RoboDK station: Example-03.b-Welding Station - Fanuc.rdk

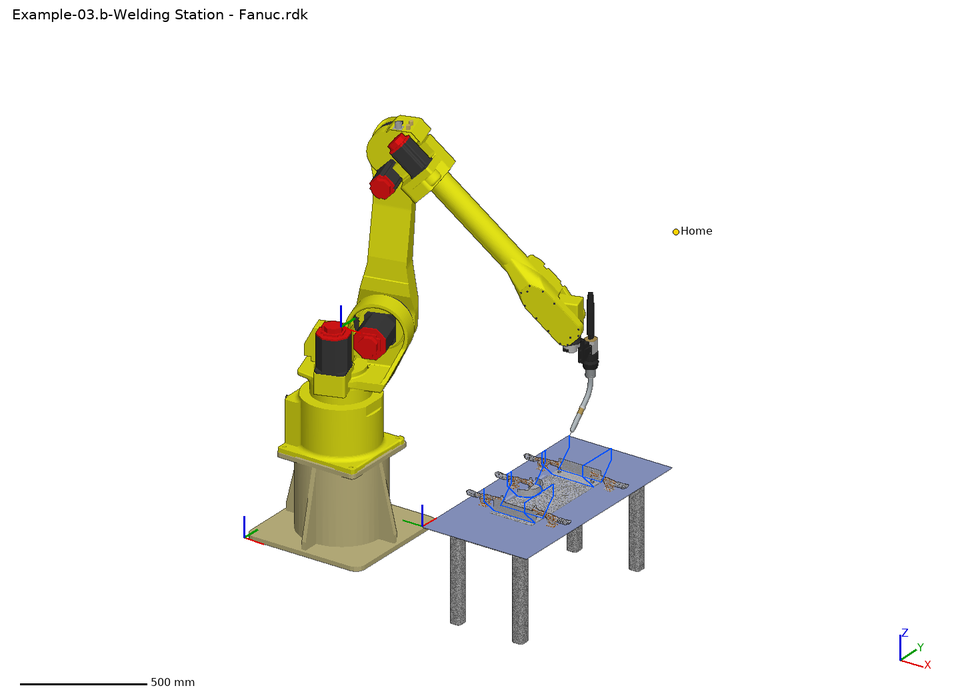
[picture v0: the station drawn from its stored meshes, robots at their saved joint values, targets as dots, program paths as lines]
Station Ex 01 - Fanuc Welding Station (saved by RoboDK 5.2.3). Poses are relative to the parent item; angles as X-Y-Z fixed-axis rotations.
Station parameters (name, value as stored): Torch1, 4, red, 0
  - frame Fanuc ARC Mate 120iB/10L Base at (0, 0, 525) mm
    - robot Fanuc ARC Mate 120iB/10L: 6 axes, payload 10 kg, reach 1885 mm, repeatability 0.1 mm, weight 225 kg
        modified DH rows (alpha deg, a mm, theta deg, d mm): 0, 0, 0, 525; -90, 150, -90, 0; 0, 770, 0, 0; -90, 100, 0, 960; 90, 0, 0, 0; -90, 0, 0, 100
        base shift (0, 0, -525) mm
        joint limits [-170, -80, -170, -200, -140, -150] to [170, 170, 250, 200, 140, 450]; home [0, 0, 0, 0, 0, 0]; saved at [18.463, 3.094, -45.099, 0, -44.901, 431.537]
      - tool Daihen OTC weld gun, TCP at (-2, 0, 402) mm, rotated rx 0 ry 45 rz 180 deg, size 201.6 x 65.1 x 567.7 mm
  - frame Table at (741.65, -500, 58.58) mm, rotated rx 0 ry 0 rz 90 deg
    - target Home (joint target) at (500, -870.35, 1334.42) mm, rotated rx -180 ry 45 rz 90 deg; joints [0, 0, 0, 0, 0, 0] of Fanuc ARC Mate 120iB/10L
    - object Weld 1 at (0, 0, 0) mm, size 1000 x 500 x 492.1 mm, geometry from Weld 1.step
  - frame World at (-274.99, -271.79, -366.75) mm
    - object Base at (0, 0, 0) mm, size 550 x 550 x 367.5 mm, geometry from Base.step
  - program Go_Home (3 instructions, listed below)
  - machining project Weld 1 Settings: rotZ(0) | rotX(0)*rotY(0) | rotz(0) | onStart | ArcStart | onApproach | onPoint | onRetract | onFinish | SetRPM(%1) | SetTool(%1) | Extruder(%1) | default | default | OutOnMov(%1) | OutOffMov(%1) | ArcEnd | M_RunCode(%1)
  - program Weld (87 instructions, listed below)
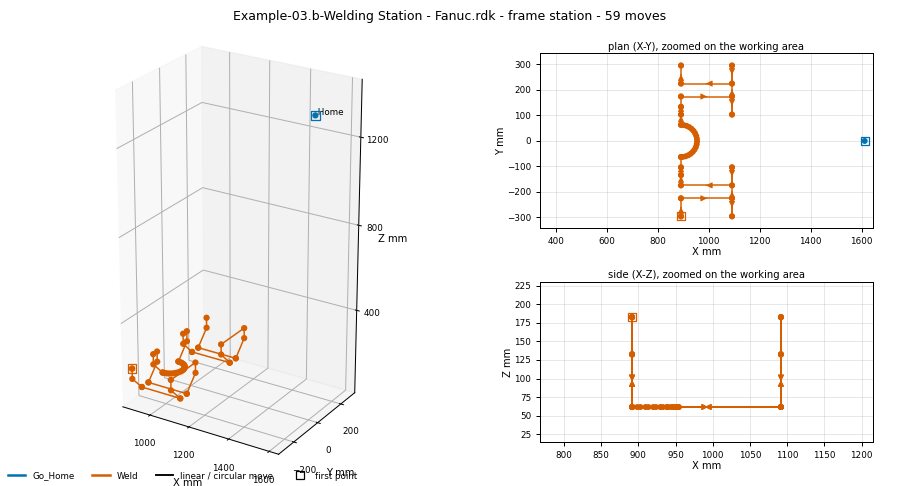
[picture p0: tool path of Example-03.b-Welding Station - Fanuc.rdk in frame station, 59 of 59 moves have a stored position in this frame; points joined in program order, loops and branches not executed]

--- program Go_Home (robot Fanuc ARC Mate 120iB/10L) ---
  Set Ref.: Table_1
  Set Tool: Daihen OTC weld gun
  MoveJ (Home)

--- program Weld (robot Fanuc ARC Mate 120iB/10L) ---
  Smooth(1)
  Set speed (1000.0 mm/s)
  Set Ref.: Table
  Set Tool: Daihen OTC weld gun
  Show Daihen OTC weld gun
  MoveJ 1 to (204.29, -150, 123.89) mm, rotated rx -180 ry -45 rz 0 deg; joints [-18.462, 3.094, -45.099, 0.004, -44.9, -71.541]
  MoveL 2 to (204.29, -150, 123.89) mm, rotated rx -180 ry -45 rz 0 deg; joints [-18.462, 3.094, -45.099, 0.004, -44.9, -71.541]
  MoveL 3 to (204.29, -150, 73.89) mm, rotated rx 180 ry -45 rz 0 deg; joints [-18.462, 6.125, -48.775, 0.004, -41.225, -71.541]
  MoveL 4 to (275, -150, 3.17) mm, rotated rx -180 ry -45 rz 0 deg; joints [-14.282, 9.561, -54.238, 0.005, -35.762, -75.722]
  Call ArcStart
  MoveL 5 to (275, -150, 3.17) mm, rotated rx -180 ry -45 rz 0 deg; joints [-14.282, 9.561, -54.238, 0.005, -35.762, -75.722]
  Set speed (50.0 mm/s)
  MoveL 6 to (275, -350, 3.17) mm, rotated rx -180 ry -45 rz 0 deg; joints [-11.745, 21.241, -50.649, 0.004, -39.351, -78.258]
  Set speed (1000.0 mm/s)
  Call ArcEnd
  MoveL 7 to (275, -350, 3.17) mm, rotated rx -180 ry -45 rz 0 deg; joints [-11.745, 21.241, -50.649, 0.004, -39.351, -78.258]
  MoveL 8 to (204.29, -350, 73.89) mm, rotated rx -180 ry -45 rz 0 deg; joints [-15.253, 18.382, -46.011, 0.004, -43.988, -74.75]
  MoveL 9 to (204.29, -350, 123.89) mm, rotated rx -180 ry -45 rz 0 deg; joints [-15.253, 15.892, -42.964, 0.004, -47.035, -74.749]
  Set speed (1000.0 mm/s)
  MoveL 10 to (396.51, -350, 124.06) mm, rotated rx -161.12 ry -41.64 rz 152.76 deg; joints [-5.087, 6.369, -45.968, 0.986, -29.938, 80.079]
  MoveL 11 to (396.51, -350, 74.06) mm, rotated rx 180 ry -45 rz -180 deg; joints [-5.311, 16.208, -46.675, 0, -43.325, 95.311]
  MoveL 12 to (325.8, -350, 3.35) mm, rotated rx -180 ry -45 rz 180 deg; joints [-8.964, 20.662, -50.867, 0, -39.133, 98.964]
  Call ArcStart
  MoveL 13 to (325.8, -350, 3.35) mm, rotated rx 180 ry -45 rz -180 deg; joints [-8.964, 20.662, -50.867, 0, -39.133, 98.964]
  Set speed (50.0 mm/s)
  MoveL 14 to (325.8, -150, 3.35) mm, rotated rx 180 ry -45 rz 180 deg; joints [-10.931, 8.786, -54.371, 0, -35.629, 100.931]
  Set speed (1000.0 mm/s)
  Call ArcEnd
  MoveL 15 to (325.8, -150, 3.35) mm, rotated rx 180 ry -45 rz 180 deg; joints [-10.931, 8.786, -54.371, 0, -35.629, 100.931]
  MoveL 16 to (396.51, -150, 74.06) mm, rotated rx 180 ry -45 rz -180 deg; joints [-6.494, 3.155, -49.022, 0, -40.978, 96.494]
  MoveL 17 to (396.51, -150, 124.06) mm, rotated rx 180 ry -45 rz -180 deg; joints [-6.494, -0.022, -45.172, 0, -44.828, 96.494]
  Set speed (1000.0 mm/s)
  MoveL 18 to (366.29, -150, 123.89) mm, rotated rx -161.12 ry -41.64 rz -27.24 deg; joints [-8.47, 9.686, -45.5, 0.389, -58.602, 264.012]
  MoveL 19 to (366.29, -150, 73.89) mm, rotated rx -180 ry -45 rz 0 deg; joints [-8.654, 3.486, -49.016, 0, -40.984, 278.654]
  MoveL 20 to (437, -150, 3.17) mm, rotated rx -180 ry -45 rz 0 deg; joints [-4.169, 7.888, -54.543, 0, -35.457, 274.169]
  Call ArcStart
  MoveL 21 to (437, -150, 3.17) mm, rotated rx -180 ry -45 rz 0 deg; joints [-4.169, 7.888, -54.543, 0, -35.457, 274.169]
  Set speed (50.0 mm/s)
  MoveL 22 to (437.39, -157.02, 3.17) mm, rotated rx -180 ry -45 rz 6.4 deg; joints [-4.11, 8.354, -54.464, 0, -35.536, 280.506]
  MoveL 23 to (439.63, -168.01, 3.17) mm, rotated rx -180 ry -45 rz 16.61 deg; joints [-3.915, 9.069, -54.333, 0, -35.667, 290.523]
  MoveL 24 to (443.78, -178.42, 3.17) mm, rotated rx 180 ry -45 rz 26.82 deg; joints [-3.604, 9.733, -54.203, 0, -35.797, 300.424]
  MoveL 25 to (449.71, -187.94, 3.17) mm, rotated rx 180 ry -45 rz 37.03 deg; joints [-3.191, 10.329, -54.079, 0, -35.921, 310.223]
  MoveL 26 to (457.23, -196.26, 3.17) mm, rotated rx -180 ry -45 rz 47.24 deg; joints [-2.689, 10.841, -53.967, 0, -36.033, 319.933]
  MoveL 27 to (466.11, -203.11, 3.17) mm, rotated rx 180 ry -45 rz 57.46 deg; joints [-2.116, 11.257, -53.872, 0, -36.128, 329.572]
  MoveL 28 to (476.06, -208.27, 3.17) mm, rotated rx 180 ry -45 rz 67.67 deg; joints [-1.486, 11.568, -53.799, 0, -36.201, 339.154]
  MoveL 29 to (486.77, -211.6, 3.17) mm, rotated rx 180 ry -45 rz 77.88 deg; joints [-0.819, 11.766, -53.751, 0, -36.249, 348.698]
  MoveL 30 to (497.9, -212.97, 3.17) mm, rotated rx 180 ry -45 rz 88.09 deg; joints [-0.13, 11.847, -53.731, 0, -36.269, 358.222]
  MoveL 31 to (509.1, -212.34, 3.17) mm, rotated rx 180 ry -45 rz 98.3 deg; joints [0.563, 11.81, -53.74, 0, -36.26, 367.741]
  MoveL 32 to (520.01, -209.74, 3.17) mm, rotated rx 180 ry -45 rz 108.52 deg; joints [1.24, 11.655, -53.778, 0, -36.222, 377.276]
  MoveL 33 to (530.28, -205.25, 3.17) mm, rotated rx 180 ry -45 rz 118.73 deg; joints [1.886, 11.386, -53.842, 0, -36.158, 386.842]
  MoveL 34 to (539.6, -199, 3.17) mm, rotated rx -180 ry -45 rz 128.94 deg; joints [2.483, 11.008, -53.929, 0, -36.071, 396.457]
  MoveL 35 to (547.66, -191.21, 3.17) mm, rotated rx 180 ry -45 rz 139.15 deg; joints [3.013, 10.531, -54.035, 0, -35.965, 406.139]
  MoveL 36 to (554.21, -182.1, 3.17) mm, rotated rx 180 ry -45 rz 149.36 deg; joints [3.461, 9.965, -54.156, 0, -35.844, 415.903]
  MoveL 37 to (559.04, -171.98, 3.17) mm, rotated rx -180 ry -45 rz 159.58 deg; joints [3.811, 9.324, -54.284, 0, -35.716, 425.765]
  MoveL 38 to (562, -161.17, 3.17) mm, rotated rx -180 ry -45 rz 169.79 deg; joints [4.051, 8.626, -54.415, 0, -35.585, 435.737]
  MoveL 39 to (563, -150, 3.17) mm, rotated rx 180 ry -45 rz -180 deg; joints [4.169, 7.888, -54.543, 0, -35.457, 445.831]
  Set speed (1000.0 mm/s)
  Call ArcEnd
  MoveL 40 to (563, -150, 3.17) mm, rotated rx 180 ry -45 rz -180 deg; joints [4.169, 7.888, -54.543, 0, -35.457, 445.831]
  MoveL 41 to (633.71, -150, 73.89) mm, rotated rx 180 ry -45 rz -180 deg; joints [8.654, 3.486, -49.016, 0, -40.984, 441.346]
  MoveL 42 to (633.71, -150, 123.89) mm, rotated rx 180 ry -45 rz -180 deg; joints [8.654, 0.324, -45.184, 0, -44.816, 441.346]
  Set speed (1000.0 mm/s)
  MoveL 43 to (603.49, -150, 124.06) mm, rotated rx 161.12 ry -41.64 rz 27.24 deg; joints [6.397, -8.748, -45.643, -0.343, -30.253, 278.092]
  MoveL 44 to (603.49, -150, 74.06) mm, rotated rx -180 ry -45 rz 0 deg; joints [6.494, 3.155, -49.022, 0, -40.978, 263.506]
  MoveL 45 to (674.2, -150, 3.35) mm, rotated rx -180 ry -45 rz 0 deg; joints [10.931, 8.786, -54.371, 0, -35.629, 259.069]
  Call ArcStart
  MoveL 46 to (674.2, -150, 3.35) mm, rotated rx -180 ry -45 rz 0 deg; joints [10.931, 8.786, -54.371, 0, -35.629, 259.069]
  Set speed (50.0 mm/s)
  MoveL 47 to (674.2, -350, 3.35) mm, rotated rx -180 ry -45 rz 0 deg; joints [8.964, 20.662, -50.867, 0, -39.133, 261.036]
  Set speed (1000.0 mm/s)
  Call ArcEnd
  MoveL 48 to (674.2, -350, 3.35) mm, rotated rx -180 ry -45 rz 0 deg; joints [8.964, 20.662, -50.867, 0, -39.133, 261.036]
  MoveL 49 to (603.49, -350, 74.06) mm, rotated rx -180 ry -45 rz 0 deg; joints [5.311, 16.208, -46.675, 0, -43.325, 264.689]
  MoveL 50 to (603.49, -350, 124.06) mm, rotated rx -180 ry -45 rz 0 deg; joints [5.311, 13.631, -43.529, 0, -46.471, 264.689]
  Set speed (1000.0 mm/s)
  MoveL 51 to (795.71, -350, 123.89) mm, rotated rx -161.12 ry -41.64 rz 152.76 deg; joints [17.86, 9.43, -45.544, 11.158, -32.112, 409.106]
  MoveL 52 to (795.71, -350, 73.89) mm, rotated rx 180 ry -45 rz -180 deg; joints [15.254, 18.383, -46.011, 0, -43.989, 434.746]
  MoveL 53 to (725, -350, 3.17) mm, rotated rx 180 ry -45 rz -180 deg; joints [11.747, 21.241, -50.649, 0, -39.351, 438.253]
  Call ArcStart
  MoveL 54 to (725, -350, 3.17) mm, rotated rx 180 ry -45 rz -180 deg; joints [11.747, 21.241, -50.649, 0, -39.351, 438.253]
  Set speed (50.0 mm/s)
  MoveL 55 to (725, -150, 3.17) mm, rotated rx 180 ry -45 rz 180 deg; joints [14.283, 9.562, -54.238, 0, -35.762, 435.717]
  Set speed (1000.0 mm/s)
  Call ArcEnd
  MoveL 56 to (725, -150, 3.17) mm, rotated rx 180 ry -45 rz 180 deg; joints [14.283, 9.562, -54.238, 0, -35.762, 435.717]
  MoveL 57 to (795.71, -150, 73.89) mm, rotated rx 180 ry -45 rz 180 deg; joints [18.463, 6.126, -48.775, 0, -41.225, 431.537]
  MoveL 58 to (795.71, -150, 123.89) mm, rotated rx -180 ry -45 rz 180 deg; joints [18.463, 3.094, -45.099, 0, -44.901, 431.537]
